// TIA Portal V16 export
// export: Created 2021-12-01T20:36:53.8748173Z, ExportSetting WithDefaults, DisplayName Totally Integrated Automation Portal, DisplayVersion V16 Update 4, DisplayName TIA Portal Version Control Interface, DisplayVersion V16 Update 2, DisplayName TIA Portal Openness, DisplayVersion V16 Update 4, DisplayName SINAMICS Startdrive Advanced, DisplayVersion V16 Update 5, DisplayName SINAMICS Startdrive G130, G150, S120, S150, SINAMICS MV, S210, DisplayVersion V16 Update 5, DisplayName SINAMICS Startdrive G110M, G120, G120C, G120D, G120P, G115D, DisplayVersion V16 Update 5, DisplayName STEP 7 Professional, DisplayVersion V16 Update 4, DisplayName STEP 7 Safety, DisplayVersion V16, DisplayName WinCC Advanced, DisplayVersion V16 Update 4
DATA_BLOCK "OPMODE09_EQUIPMENT_DATA_FB_IDB"   // DB247
AUTHOR : Tesla
FAMILY : Data
VERSION : 0.1
// stored: AssignedProDiagFB OPMODE09_PD, AutoNumber false, DBAccessibleFromOPCUA true, InstanceOfName EQUIPMENT_DATA_FB, InstanceOfType FB
"EQUIPMENT_DATA_FB"
   // VAR_INPUT
   //    EQUIPMENT_NAME { ExternalAccessible := 'False'; ExternalVisible := 'False'; ExternalWritable := 'False'} : String;
   //    MODULE_NAME { ExternalAccessible := 'False'; ExternalVisible := 'False'; ExternalWritable := 'False'} : String;
   //    UTC_DATETIME { ExternalAccessible := 'False'; ExternalVisible := 'False'; ExternalWritable := 'False'} : DTL;
   //    AUTOMATIC { ExternalAccessible := 'False'; ExternalVisible := 'False'; ExternalWritable := 'False'} : Bool;
   //    MANUAL { ExternalAccessible := 'False'; ExternalVisible := 'False'; ExternalWritable := 'False'} : Bool;
   //    ENGINEERING { ExternalAccessible := 'False'; ExternalVisible := 'False'; ExternalWritable := 'False'} : Bool;
   //    SETUP { ExternalAccessible := 'False'; ExternalVisible := 'False'; ExternalWritable := 'False'} : Bool;
   //    NON_SCHEDULED_TIME { ExternalAccessible := 'False'; ExternalVisible := 'False'; ExternalWritable := 'False'} : Bool;
   //    HOMING { ExternalAccessible := 'False'; ExternalVisible := 'False'; ExternalWritable := 'False'} : Bool;
   //    HOMED { ExternalAccessible := 'False'; ExternalVisible := 'False'; ExternalWritable := 'False'} : Bool;
   //    ABORTING { ExternalAccessible := 'False'; ExternalVisible := 'False'; ExternalWritable := 'False'} : Bool;
   //    ABORTED { ExternalAccessible := 'False'; ExternalVisible := 'False'; ExternalWritable := 'False'} : Bool;
   //    PAUSING { ExternalAccessible := 'False'; ExternalVisible := 'False'; ExternalWritable := 'False'} : Bool;
   //    PAUSED { ExternalAccessible := 'False'; ExternalVisible := 'False'; ExternalWritable := 'False'} : Bool;
   //    STOPPING { ExternalAccessible := 'False'; ExternalVisible := 'False'; ExternalWritable := 'False'} : Bool;
   //    STOPPED { ExternalAccessible := 'False'; ExternalVisible := 'False'; ExternalWritable := 'False'} : Bool;
   //    CYCLE_RUNNING { ExternalAccessible := 'False'; ExternalVisible := 'False'; ExternalWritable := 'False'} : Bool;
   //    FAULTED { ExternalAccessible := 'False'; ExternalVisible := 'False'; ExternalWritable := 'False'} : Bool;
   //    BLOCKED { ExternalAccessible := 'False'; ExternalVisible := 'False'; ExternalWritable := 'False'} : Bool;
   //    STARVED { ExternalAccessible := 'False'; ExternalVisible := 'False'; ExternalWritable := 'False'} : Bool;
   //    REASON { ExternalAccessible := 'False'; ExternalVisible := 'False'; ExternalWritable := 'False'} : DInt;
   //    PART_ID { ExternalAccessible := 'False'; ExternalVisible := 'False'; ExternalWritable := 'False'} : String;
   //    CARRIER_ID { ExternalAccessible := 'False'; ExternalVisible := 'False'; ExternalWritable := 'False'} : String;
   //    PALLET_ID { ExternalAccessible := 'False'; ExternalVisible := 'False'; ExternalWritable := 'False'} : String;
   //    TARGET_CYCLE_TIME { ExternalAccessible := 'False'; ExternalVisible := 'False'; ExternalWritable := 'False'} : Time;
   //    "ENABLE_NON-SCHEDULED_TIME" { ExternalAccessible := 'False'; ExternalVisible := 'False'; ExternalWritable := 'False'} : Bool;
   //    ENABLE_CYCLE_TIME { ExternalAccessible := 'False'; ExternalVisible := 'False'; ExternalWritable := 'False'} : Bool;
   //    SHIFT_COUNT { ExternalAccessible := 'False'; ExternalVisible := 'False'; ExternalWritable := 'False'} : DInt;
   //    CURRENT_STEP_HISTORY { ExternalAccessible := 'False'; ExternalVisible := 'False'; ExternalWritable := 'False'} : Array[0.."EQUIPMENTDATA_STEPHISTORYLENGTH"] of "GRAPH_STEP_HISTORY_UDT";
   //    ACTIVE_ALARMS { ExternalAccessible := 'False'; ExternalVisible := 'False'; ExternalWritable := 'False'} : Array[0.."EQUIPMENTDATA_ACTIVEALARMSLENGTH"] of "ALARM_DATA_UDT";
   //    BUFFER1_MAX_COUNT : DInt;
   //    BUFFER1_MIN_COUNT : DInt;
   //    BUFFER1_ACTUAL_COUNT : DInt;
   //    BUFFER2_MAX_COUNT : DInt;
   //    BUFFER2_MIN_COUNT : DInt;
   //    BUFFER2_ACTUAL_COUNT : DInt;
   // END_VAR
   // VAR_OUTPUT
   //    CYCLE_TIMER_RUN { ExternalAccessible := 'False'; ExternalVisible := 'False'; ExternalWritable := 'False'} : Bool;
   //    CYCLE_TIMER_HOLD { ExternalAccessible := 'False'; ExternalVisible := 'False'; ExternalWritable := 'False'} : Bool;
   //    CURRENT_CYCLE_DURATION { ExternalAccessible := 'False'; ExternalVisible := 'False'; ExternalWritable := 'False'} : Time;
   //    CURRENT_STATE_DURATION { ExternalAccessible := 'False'; ExternalVisible := 'False'; ExternalWritable := 'False'} : Time;
   //    CURRENT_SHIFT_COUNT { ExternalAccessible := 'False'; ExternalVisible := 'False'; ExternalWritable := 'False'} : DInt;
   //    CURRENT_BUFFER1_MAX_COUNT { ExternalAccessible := 'False'; ExternalVisible := 'False'; ExternalWritable := 'False'} : DInt;
   //    CURRENT_BUFFER1_MIN_COUNT { ExternalAccessible := 'False'; ExternalVisible := 'False'; ExternalWritable := 'False'} : DInt;
   //    CURRENT_BUFFER1_ACTUAL_COUNT { ExternalAccessible := 'False'; ExternalVisible := 'False'; ExternalWritable := 'False'} : DInt;
   //    CURRENT_BUFFER2_MAX_COUNT { ExternalAccessible := 'False'; ExternalVisible := 'False'; ExternalWritable := 'False'} : DInt;
   //    CURRENT_BUFFER2_MIN_COUNT : DInt;
   //    CURRENT_BUFFER2_ACTUAL_COUNT : DInt;
   // END_VAR
   // VAR_IN_OUT
   //    HMI_SCADA : "EQUIPMENT_DATA_OUT_UDT";
   // END_VAR
   // VAR
   //    AX_EndOfCycleOld { ExternalAccessible := 'False'; ExternalVisible := 'False'; ExternalWritable := 'False'} : Bool;
   //    AX_StoppedOld { ExternalAccessible := 'False'; ExternalVisible := 'False'; ExternalWritable := 'False'} : Bool;
   //    AX_EndOfCycleTrigger { ExternalAccessible := 'False'; ExternalVisible := 'False'; ExternalWritable := 'False'} : Bool;
   //    AX_CycleRunOld { ExternalAccessible := 'False'; ExternalVisible := 'False'; ExternalWritable := 'False'} : Bool;
   //    AX_CycleStart { ExternalAccessible := 'False'; ExternalVisible := 'False'; ExternalWritable := 'False'} : Bool;
   // END_VAR
   // VAR RETAIN
   //    CycleCounter { ExternalAccessible := 'False'; ExternalVisible := 'False'; ExternalWritable := 'False'} : UInt;
   //    CycleTimer { ExternalAccessible := 'False'; ExternalVisible := 'False'; ExternalWritable := 'False'} : TONR_TIME;
   //    Elapsed { ExternalAccessible := 'False'; ExternalVisible := 'False'; ExternalWritable := 'False'} : Time;
   // END_VAR
   // VAR
   //    DelayTimer { ExternalAccessible := 'False'; ExternalVisible := 'False'; ExternalWritable := 'False'} : Array[0..10] of Time;
   //    DelayTMR { ExternalAccessible := 'False'; ExternalVisible := 'False'; ExternalWritable := 'False'} : Array[0..9] of TON_TIME;
   // END_VAR
   // VAR RETAIN
   //    PrevState { ExternalAccessible := 'False'; ExternalVisible := 'False'; ExternalWritable := 'False'} : "EQUIPMENT_STATE_UDT";
   // END_VAR
   // VAR
   //    AX_EndOfCycleTriggerDelayed { ExternalAccessible := 'False'; ExternalVisible := 'False'; ExternalWritable := 'False'} : Bool;
   // END_VAR
BEGIN
END_DATA_BLOCK
